// TIA Portal V18 export
FUNCTION "Math" : Void   // FC3, LAD
{ S7_Optimized_Access := 'TRUE' }
// stored: SetENOAutomatically false
   VAR_TEMP
      RetVal : Int;
   END_VAR
BEGIN

REGION Network 1
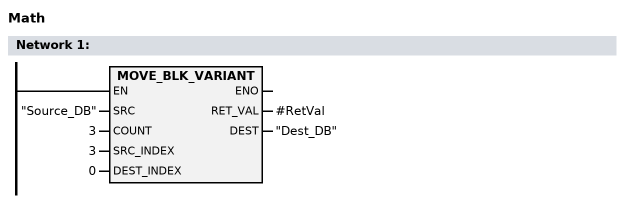
   RUNG wire#powerrail
      MOVE_BLK_VARIANT(SRC := "Source_DB", COUNT := 3, SRC_INDEX := 3, DEST_INDEX := 0, Ret_Val => #RetVal, DEST => "Dest_DB")
   END_RUNG
   // the same network as SCL:
   #RetVal := MOVE_BLK_VARIANT(SRC := "Source_DB",
                           COUNT := 3,
                           SRC_INDEX := 3,
                           DEST_INDEX := 0,
                           DEST => "Dest_DB");
END_REGION
END_FUNCTION
